(* Logix 5000 project; controller Ex_2_06 Emulate 5570 rev 33.11; software revision 33.00 *)
// Turn on and off lamps with a push button

TASK MainTask (continuous, watchdog 500 ms) : MainProgram

MODULES
   Local : Emulate 5570 (ICP 4, rev 33.11)
END_MODULES

VAR_GLOBAL   (* controller tags *)
   P1 : BOOL;   // Lamp_P1
   P2 : BOOL;   // Lamp_P2
   S1 : BOOL;   // Push Button S1
END_VAR

PROGRAM MainProgram   (* main routine MainRoutine *)

ROUTINE MainRoutine   (* ladder *)
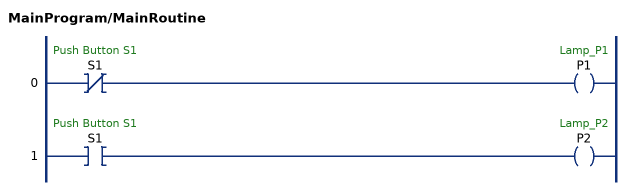
   0: XIO(S1)OTE(P1);
   1: XIC(S1)OTE(P2);
END_ROUTINE
END_PROGRAM
